PROGRAM P_Demo_FB_BARBlindPositionEntry
VAR
    fb : FB_BARBlindPositionEntry;                            // 被演示 FB 实例
    eDataSecurityType_in : E_HVACDataSecurityType ;
    bSetDefault_in : BOOL := FALSE;
    lrSunElevation1_io : REAL := 0.0;
    uiBlindPosition1_io : UINT := 0;
    lrSunElevation2_io : REAL := 0.0;
    uiBlindPosition2_io : UINT := 0;
    lrSunElevation3_io : REAL := 0.0;
    uiBlindPosition3_io : UINT := 0;
    lrSunElevation4_io : REAL := 0.0;
    uiBlindPosition4_io : UINT := 0;
    bValid_out : BOOL;
    uiErrorId_out : UDINT;
    stBlindPositionTable_out : ST_BARBlindPositionTable;
END_VAR

// ============================================================================
// Tc2_HVAC.FB_BARBlindPositionEntry 演示程序
// ============================================================================
// 场景：把本 FB 实例化到一个 PLC 程序里，每周期单次调用；按需要把 VAR_INPUT 与
//       VAR_IN_OUT 接到工程信号；VAR_OUTPUT 写入对应监视变量。
// 价值：使用本 FB 比手写状态机 / 控制算法节省大量代码；与 Tc2_HVAC 体系内其它 FB
//       直接对接，命名 / 持久化 / 模式仲裁等约定一致。具体语义见 FB_BARBlindPositionEntry.md 主文档。
// 验证步骤：
//   1. 右键 PLC 项目下 POUs 文件夹 → Add → Existing Item → 选本 .TcPOU 文件
//   2. 引用 Tc2_HVAC（References → Add library）
//   3. 编译 → 登录 → 运行
//   4. 在线写各 *_in 输入信号触发 FB；在线 monitor *_out 引脚观察状态
// ============================================================================

fb(
    eDataSecurityType := eDataSecurityType_in,
    bSetDefault := bSetDefault_in,
    lrSunElevation1 := lrSunElevation1_io,
    uiBlindPosition1 := uiBlindPosition1_io,
    lrSunElevation2 := lrSunElevation2_io,
    uiBlindPosition2 := uiBlindPosition2_io,
    lrSunElevation3 := lrSunElevation3_io,
    uiBlindPosition3 := uiBlindPosition3_io,
    lrSunElevation4 := lrSunElevation4_io,
    uiBlindPosition4 := uiBlindPosition4_io,
    bValid => bValid_out,
    uiErrorId => uiErrorId_out,
    stBlindPositionTable => stBlindPositionTable_out
);

END_PROGRAM

(* stored: Version 1.1.0.1, ProductVersion 3.1.4024.5
   POU P_Demo_FB_BARBlindPositionEntry: Id {61624939-b06d-5ff4-8a66-3c2678b5fea3}, SpecialFunc None *)
